FUNCTION_BLOCK FB_FMS205_SFC
VAR_INPUT
	ctInp		: S_ControllerInput;
	FinCiclo	: BOOL;
	IC			: BOOL;
	//EmpProducir: BOOL; // se pide a la fms205 que empiece a producr
	//DejProducir: BOOL; // se pide a la fms205 que deje de producir 
	
	//EmpRestaurar: BOOL; // se pide a la fms205 que hay que empezar restaurar
	//DejRestaurar: BOOL; // se pide a la fms205 que deje de restaurar 
END_VAR
VAR_OUTPUT
	HayProducir: BOOL;  // la fms205 indica a los módulos que hay que producir
	HayRestaurar: BOOL; // la fms205 indica a los módulos que hay que restaurar
	Hecho: BOOL; // la fms205 informa al director que ha hecho lo que se le ha pedidod
END_VAR
VAR
END_VAR

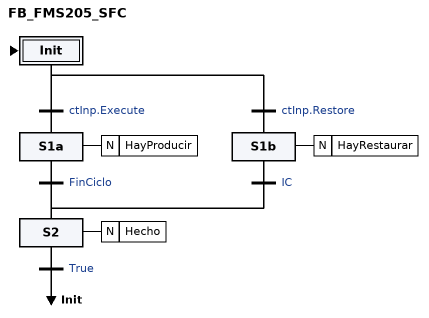
INITIAL_STEP Init:
END_STEP
TRANSITION FROM Init TO S1a
    := ctInp.Execute;
END_TRANSITION
STEP S1a:
    HayProducir(N);
END_STEP
TRANSITION FROM S1a TO S2
    := FinCiclo;
END_TRANSITION
TRANSITION FROM Init TO S1b
    := ctInp.Restore;
END_TRANSITION
STEP S1b:
    HayRestaurar(N);
END_STEP
TRANSITION FROM S1b TO S2
    := IC;
END_TRANSITION
STEP S2:
    Hecho(N);
END_STEP
TRANSITION FROM S2 TO Init
    := True;
END_TRANSITION

END_FUNCTION_BLOCK

(* stored: Version 1.1.0.1, ProductVersion 3.1.4024.11
   POU FB_FMS205_SFC: Id {e9cd1dca-e7a6-4d28-ad92-4284024c4317}, SpecialFunc None *)
